// E_PIDMode
// Rev 1.0 - October 23, 2024

TYPE E_PIDMode :
(
	eOff						:= 0,
	eManual,
	eAuto,
	eTune
);
END_TYPE

(* stored: Version 1.1.0.1, ProductVersion 3.1.4024.13
   DUT E_PIDMode: Id {c4cf29d1-ea67-493e-88ab-c791fbb776d9} *)
